ADAPTER TestAdapter (* Adapter Interface *)
  (* Standard: 61499-1; Description: Copyright (c) 2019 Jan Holzweber This program and the accompanying materials are made available under the terms of the Eclipse Public License 2.0 which is available at https://www.eclipse.org/legal/epl-2.0/ SPDX-License-Identifier: EPL-2.0 *)
  (* Version 0.0, 2008-04-22, GE, 4DIAC-Consortium *)
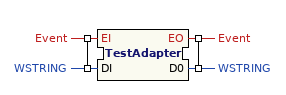
  EVENT_INPUT
    EI WITH DI; (* Request from Socket *)
  END_EVENT
  EVENT_OUTPUT
    EO WITH D0; (* Confirmation from Plug *)
  END_EVENT
  VAR_INPUT
    DI : WSTRING; (* Request Data from Socket *)
  END_VAR
  VAR_OUTPUT
    D0 : WSTRING; (* Confirmation Data from Plug *)
  END_VAR
  SERVICE SOCKET/PLUG (* Adapter Interface *)
    SEQUENCE request_confirm
      SOCKET.REQ(REQD) -> PLUG.REQ(REQD);
      PLUG.CNF(CNFD) -> SOCKET.CNF(CNFD);
    END_SEQUENCE
    SEQUENCE indication_response
      PLUG.IND(INDD) -> SOCKET.IND(INDD);
      SOCKET.RSP(RSPD) -> PLUG.RSP(RSPD);
    END_SEQUENCE
  END_SERVICE
END_ADAPTER
